FUNCTION_BLOCK FB_ManualControl IMPLEMENTS  I_ManualControl
VAR_INPUT
END_VAR
VAR_OUTPUT
END_VAR
VAR
	TEMP_1 : BOOL;
	Counter : INT;
	TEMP : BOOL;

	
END_VAR

{warning 'add method implementation '}
METHOD M_RunPump : BOOL
VAR_INPUT
	bStart	: BOOL;
	NTimes : INT;

END_VAR
VAR
	
END_VAR

IF NTimes <> 0 THEN
	IF TRUE THEN
	Counter := Counter + 1;
	END_IF
	IF Counter >= (100/(2*NTimes)) THEN
		TEMP := TRUE;
	ELSE
		TEMP := FALSE;
	END_IF
	IF Counter >= (200/(2*NTimes)) THEN
		Counter := 0;
	END_IF
ELSE
	RETURN;
END_IF

IF bstart THEN
	M_RunPump := TEMP;
ELSE
	M_RunPump := FALSE;
END_IF
END_METHOD

{warning 'add method implementation '}
METHOD M_RunValve : BOOL
VAR_INPUT
	bStart	: BOOL;
END_VAR
VAR
	
END_VAR
M_RunValve := bStart;
END_METHOD

END_FUNCTION_BLOCK

(* stored: Version 1.1.0.1, ProductVersion 3.1.4024.6
   POU FB_ManualControl: Id {bff1fefb-ba76-459a-a178-e043564c529d}, SpecialFunc None
   Method M_RunPump: Id {694dc806-2681-4d62-ae30-ad2094a5807a}
   Method M_RunValve: Id {b1fc87d9-3aaf-4b10-a767-42345da696c4} *)
